FUNCTION_BLOCK FB_ControlElement_HMI EXTENDS FB_BaseControlElement_HMI IMPLEMENTS ITF_ControlElement_HMI
VAR
	itfControlElementConnector			: ITF_ControlElement_HMI_Connector;
	refstControlElementData				: REFERENCE TO ST_ControlElement_HMI;
END_VAR

END_FUNCTION_BLOCK

(* stored: Version 1.1.0.1, ProductVersion 3.1.4024.15
   POU FB_ControlElement_HMI: Id {6ebe5482-b91b-4d08-bc26-129cdd0cb96c}, SpecialFunc None *)
